// TIA Portal project "INDEXING STATION" (V16)

(* hardware
DEVICE "S7-1200 station_1"  S7-1200 Station
   slot 0: "Rack_0"  S7-1200 Rack  Rack  V1.0
   slot 1: "plc1"  CPU 1214C DC/DC/DC  6ES7 214-1AG40-0XB0  V4.4
DEVICE "ET 200SP station_1"  ET 200SP-Station
   slot 0: "Rack_0"  Rack  6ES5 710-8MAx1
   slot 0: "IO device_1"  IM 155-6 PN/2 HF  6ES7 155-6AU01-0CN0  V4.2
   slot 1: "DI 8x24VDC HF_1"  DI 8x24VDC HF  6ES7 131-6BF00-0CA0  V2.0
      slot 1: "DI 8x24VDC HF_1"  DI 8x24VDC HF
   slot 2: "DI 8x24VDC HF_2"  DI 8x24VDC HF  6ES7 131-6BF00-0CA0  V2.0
      slot 1: "DI 8x24VDC HF_2"  DI 8x24VDC HF
   slot 3: "DI 8x24VDC HF_3"  DI 8x24VDC HF  6ES7 131-6BF00-0CA0  V2.0
      slot 1: "DI 8x24VDC HF_3"  DI 8x24VDC HF
   slot 4: "DQ 8x24VDC/0.5A HF_1"  DQ 8x24VDC/0.5A HF  6ES7 132-6BF00-0CA0  V2.0
      slot 1: "DQ 8x24VDC/0.5A HF_1"  DQ 8x24VDC/0.5A HF
   slot 5: "DQ 8x24VDC/0.5A HF_2"  DQ 8x24VDC/0.5A HF  6ES7 132-6BF00-0CA0  V2.0
      slot 1: "DQ 8x24VDC/0.5A HF_2"  DQ 8x24VDC/0.5A HF
   slot 6: "Server module_1"  Server module  6ES7 193-6PA00-0AA0  V1.1
      slot 1: "Server module_1"  Server module
   slot 127: "BA 2xRJ45"  BA 2xRJ45  6ES7 193-6AR00-0AA0  V0.0
      slot 1: "Port_1"  X1 P1 R  6ES7 193-6AR00-0AA0  V0.0
      slot 2: "Port_2"  X1 P2 R  6ES7 193-6AR00-0AA0  V0.0
*)

// ===== PLC "plc1"  CPU 1214C DC/DC/DC =====

VAR_GLOBAL   // PLC tag table "INPUTS&OUTPUTS_1"
   "S3_START" AT %I0.0 : Bool;
   "S4_STOP" AT %I0.1 : Bool;
   "S5_EMERGENCY_STOP" AT %I0.2 : Bool;
   "S2_OUTPUT_POWER" AT %I0.3 : Bool;
   "S6_RESET" AT %I1.0 : Bool;
   "S_AUTO" AT %I1.1 : Bool;
   "4B1_TRANSFER_CYLINDER_RETRACTED" AT %I1.2 : Bool;
   "4B2_TRANSFER_CYLINDER_EXTENDED" AT %I1.3 : Bool;
   "1B1_LIFT_CYLINDER_RETRACTED" AT %I1.4 : Bool;
   "1B2_LIFT_CYLINDER_EXTENDED" AT %I1.5 : Bool;
   "B3_PART_PRESENT(ORIENTATION_POSITION)" AT %I2.1 : Bool;
   "2B1_ROTATION_CYLINDER_RETRACTED" AT %I2.2 : Bool;
   "2B2_ROTATION_CYLINDER_EXTENDED" AT %I2.3 : Bool;
   "B2_SPOOL_UPPER_PORT" AT %I2.4 : Bool;
   "B4_INDEX_TABLE_HOME" AT %I2.5 : Bool;
   "B5_STEPPER_READY" AT %I2.6 : Bool;
   "B1_PART_PRESENT(INITIAL_POSITION)" AT %I2.7 : Bool;
   "H3_GREEN_ON" AT %Q4.0 : Bool;
   "4M1_EXTEND_TRANSFER" AT %Q4.5 : Bool;
   "1M1_EXTEND_LIFT" AT %Q4.6 : Bool;
   "1M2_RETRACT_LIFT" AT %Q4.7 : Bool;
   "M1_45_STEPPER" AT %Q5.2 : Bool;
   "M1_90_STEPPER" AT %Q5.3 : Bool;
   "3M1_RELEASE_GRIPPER" AT %Q5.4 : Bool;
   "3M2_CLOSE_GRIPPER" AT %Q5.5 : Bool;
   "2M1_EXTEND_ROTATION_CYLINDER" AT %Q5.6 : Bool;
   "2M2_RETRACT_ROTATION_CYLINDER" AT %Q5.7 : Bool;
   "AUTO_MEM" AT %M1.0 : Bool;
   "STOP_MEM" AT %M1.1 : Bool;
   "STEP_2_MEM_ON" AT %M1.2 : Bool;
   "STEP_3&7_MEM_ON" AT %M1.3 : Bool;
   "STEP_4_MEM_ON" AT %M1.4 : Bool;
   "MANUAL_MEM" AT %M1.5 : Bool;
   "STEPPER MEMORY 1" AT %M100.0 : Bool;
   "SM 2" AT %M100.1 : Bool;
   "SM 3" AT %M100.2 : Bool;
   "SM 4" AT %M100.3 : Bool;
   "PART_MEM" AT %M100.4 : Bool;
END_VAR

DATA_BLOCK "STEPS"   // DB1
{ S7_Optimized_Access := 'FALSE' }
VERSION : 0.1
   VAR
      "Current steps" : Int;
   END_VAR
BEGIN
END_DATA_BLOCK

ORGANIZATION_BLOCK "Main"   // OB1, LAD, ProgramCycle
TITLE = "Main Program Sweep (Cycle)"
{ S7_Optimized_Access := 'TRUE' }
VERSION : 0.1
   VAR_INPUT
      Initial_Call : Bool;   // Initial call of this OB
      Remanence : Bool;   // =True, if remanent data are available
   END_VAR
   VAR_TEMP   // added for the SCL form of the ladder/FBD networks
      _w1 : Bool;
   END_VAR
BEGIN

REGION Network 2: START LED ON
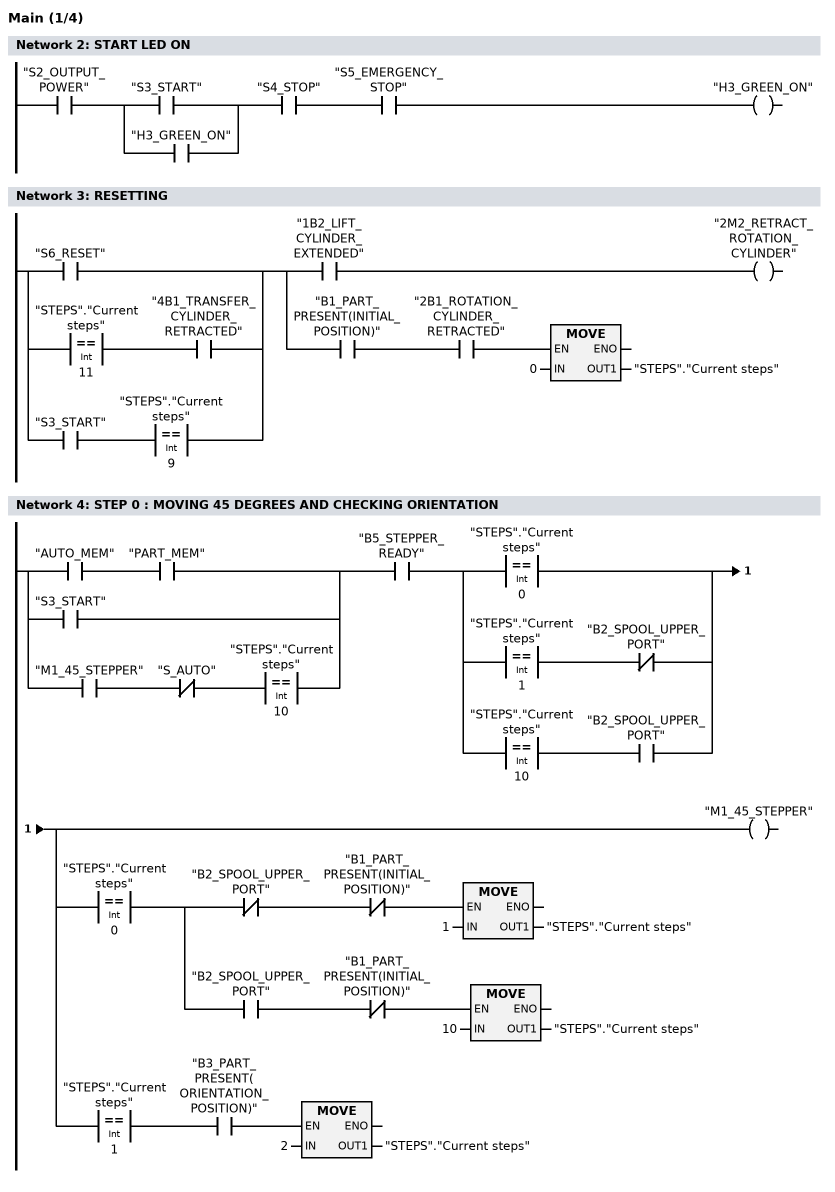
   RUNG wire#powerrail
      Contact( "S2_OUTPUT_POWER" )
      wire#w1
      Contact( "S3_START" )
      wire#w2
      Contact( "S4_STOP" )
      Contact( "S5_EMERGENCY_STOP" )
      Coil( "H3_GREEN_ON" )
   END_RUNG
   RUNG wire#w1
      Contact( "H3_GREEN_ON" )
   END_RUNG wire#w2
   // the same network as SCL:
   "H3_GREEN_ON" := "S2_OUTPUT_POWER" AND ("S3_START" OR "H3_GREEN_ON") AND "S4_STOP" AND "S5_EMERGENCY_STOP";
END_REGION

REGION Network 3: RESETTING
   RUNG wire#powerrail
      Contact( "S6_RESET" )
      wire#w1
      Contact( "1B2_LIFT_CYLINDER_EXTENDED" )
      Coil( "2M2_RETRACT_ROTATION_CYLINDER" )
   END_RUNG
   RUNG wire#powerrail
      { S7_Templates := "SrcType := Int" } EQ_Contact(in1 := "STEPS"."Current steps", in2 := 11)
      Contact( "4B1_TRANSFER_CYLINDER_RETRACTED" )
   END_RUNG wire#w1
   RUNG wire#powerrail
      Contact( "S3_START" )
      { S7_Templates := "SrcType := Int" } EQ_Contact(in1 := "STEPS"."Current steps", in2 := 9)
   END_RUNG wire#w1
   RUNG wire#w1
      Contact( "B1_PART_PRESENT(INITIAL_POSITION)" )
      Contact( "2B1_ROTATION_CYLINDER_RETRACTED" )
      { S7_GenerateENO := "TRUE" } Move(in := 0, out1 => "STEPS"."Current steps")
   END_RUNG
   // the same network as SCL:
   #_w1 := "S6_RESET" OR (("STEPS"."Current steps" = 11) AND "4B1_TRANSFER_CYLINDER_RETRACTED") OR ("S3_START" AND ("STEPS"."Current steps" = 9));
   "2M2_RETRACT_ROTATION_CYLINDER" := #_w1 AND "1B2_LIFT_CYLINDER_EXTENDED";
   IF #_w1 AND "B1_PART_PRESENT(INITIAL_POSITION)" AND "2B1_ROTATION_CYLINDER_RETRACTED" THEN
       "STEPS"."Current steps" := 0;
   END_IF;
END_REGION

REGION Network 4: STEP 0 : MOVING 45 DEGREES AND CHECKING ORIENTATION
   RUNG wire#powerrail
      Contact( "AUTO_MEM" )
      Contact( "PART_MEM" )
      wire#w1
      Contact( "B5_STEPPER_READY" )
      wire#w2
      { S7_Templates := "SrcType := Int" } EQ_Contact(in1 := "STEPS"."Current steps", in2 := 0)
      wire#w3
      Coil( "M1_45_STEPPER" )
   END_RUNG
   RUNG wire#powerrail
      Contact( "S3_START" )
   END_RUNG wire#w1
   RUNG wire#powerrail
      Contact( "M1_45_STEPPER" )
      I_Contact( "S_AUTO" )
      { S7_Templates := "SrcType := Int" } EQ_Contact(in1 := "STEPS"."Current steps", in2 := 10)
   END_RUNG wire#w1
   RUNG wire#w2
      { S7_Templates := "SrcType := Int" } EQ_Contact(in1 := "STEPS"."Current steps", in2 := 1)
      I_Contact( "B2_SPOOL_UPPER_PORT" )
   END_RUNG wire#w3
   RUNG wire#w2
      { S7_Templates := "SrcType := Int" } EQ_Contact(in1 := "STEPS"."Current steps", in2 := 10)
      Contact( "B2_SPOOL_UPPER_PORT" )
   END_RUNG wire#w3
   RUNG wire#w3
      { S7_Templates := "SrcType := Int" } EQ_Contact(in1 := "STEPS"."Current steps", in2 := 0)
      wire#w4
      I_Contact( "B2_SPOOL_UPPER_PORT" )
      I_Contact( "B1_PART_PRESENT(INITIAL_POSITION)" )
      { S7_GenerateENO := "TRUE" } Move(in := 1, out1 => "STEPS"."Current steps")
   END_RUNG
   RUNG wire#w4
      Contact( "B2_SPOOL_UPPER_PORT" )
      I_Contact( "B1_PART_PRESENT(INITIAL_POSITION)" )
      { S7_GenerateENO := "TRUE" } Move(in := 10, out1 => "STEPS"."Current steps")
   END_RUNG
   RUNG wire#w3
      { S7_Templates := "SrcType := Int" } EQ_Contact(in1 := "STEPS"."Current steps", in2 := 1)
      Contact( "B3_PART_PRESENT(ORIENTATION_POSITION)" )
      { S7_GenerateENO := "TRUE" } Move(in := 2, out1 => "STEPS"."Current steps")
   END_RUNG
   // the same network as SCL:
   "M1_45_STEPPER" := (("AUTO_MEM" AND "PART_MEM") OR "S3_START" OR ("M1_45_STEPPER" AND NOT "S_AUTO" AND ("STEPS"."Current steps" = 10))) AND "B5_STEPPER_READY" AND (("STEPS"."Current steps" = 0) OR (("STEPS"."Current steps" = 1) AND NOT "B2_SPOOL_UPPER_PORT") OR (("STEPS"."Current steps" = 10) AND "B2_SPOOL_UPPER_PORT"));
   #_w1 := "M1_45_STEPPER" AND ("STEPS"."Current steps" = 0);
   IF #_w1 AND NOT "B2_SPOOL_UPPER_PORT" AND NOT "B1_PART_PRESENT(INITIAL_POSITION)" THEN
       "STEPS"."Current steps" := 1;
   END_IF;
   IF #_w1 AND "B2_SPOOL_UPPER_PORT" AND NOT "B1_PART_PRESENT(INITIAL_POSITION)" THEN
       "STEPS"."Current steps" := 10;
   END_IF;
   IF "M1_45_STEPPER" AND ("STEPS"."Current steps" = 1) AND "B3_PART_PRESENT(ORIENTATION_POSITION)" THEN
       "STEPS"."Current steps" := 2;
   END_IF;
END_REGION

REGION Network 5: AUTOMATIC_MODE
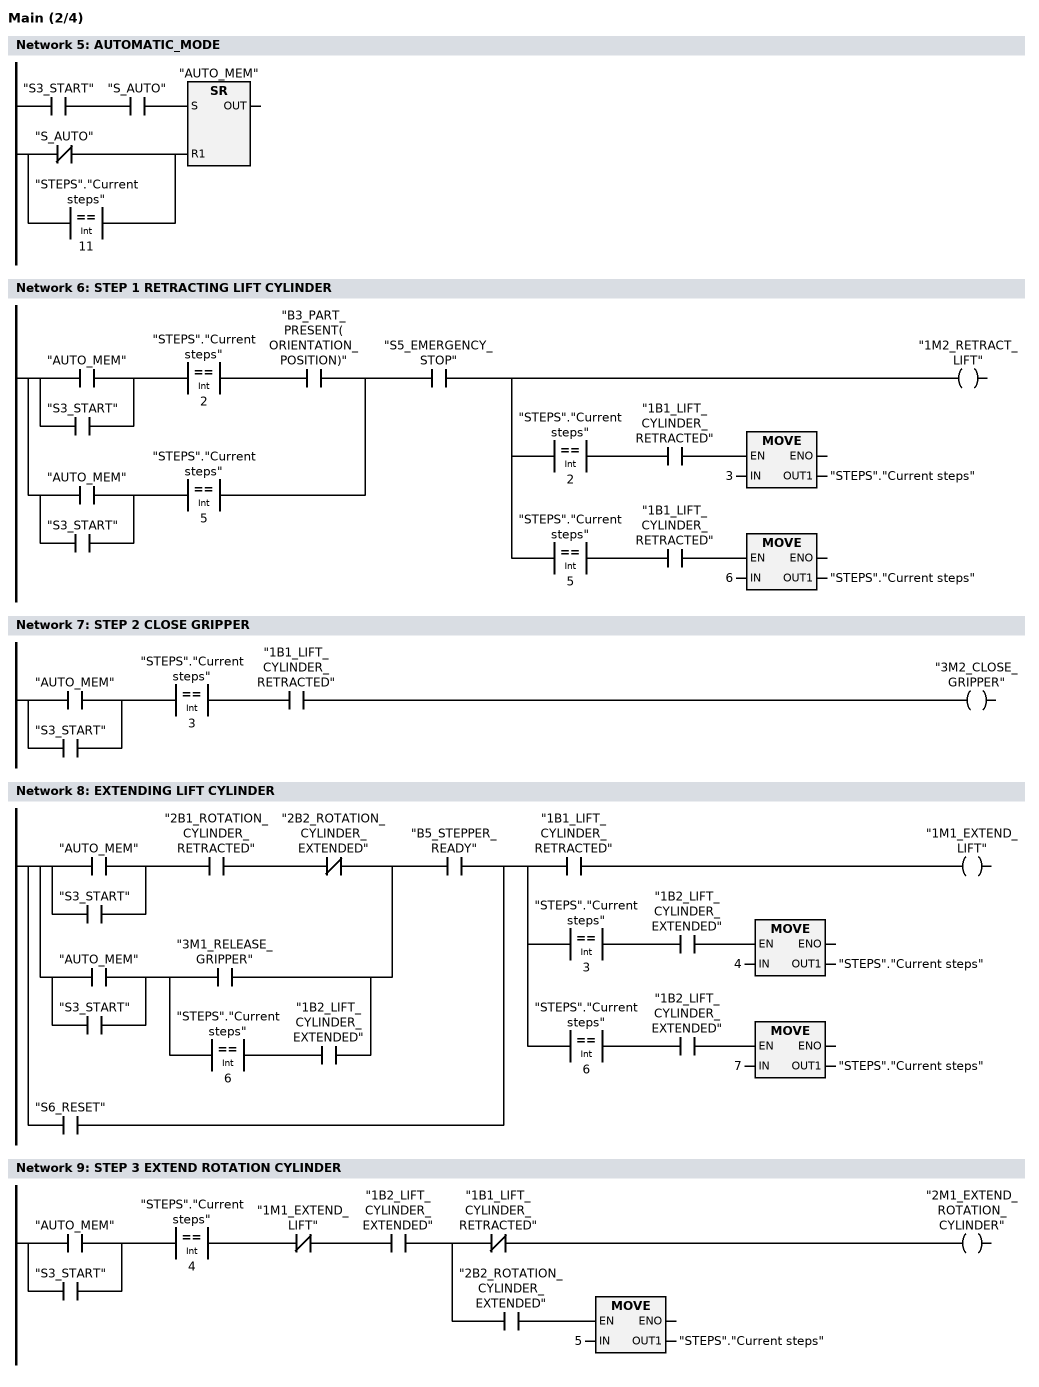
   RUNG wire#powerrail
      Contact( "S3_START" )
      Contact( "S_AUTO" )
      S_SR(operand := "AUTO_MEM", r1 := wire#w1)
   END_RUNG
   RUNG wire#powerrail
      I_Contact( "S_AUTO" )
   END_RUNG wire#w1
   RUNG wire#powerrail
      { S7_Templates := "SrcType := Int" } EQ_Contact(in1 := "STEPS"."Current steps", in2 := 11)
   END_RUNG wire#w1
   // the same network as SCL:
   IF "S3_START" AND "S_AUTO" THEN
       "AUTO_MEM" := TRUE;   // SR flip-flop
   END_IF;
   IF NOT "S_AUTO" OR ("STEPS"."Current steps" = 11) THEN "AUTO_MEM" := FALSE; END_IF;
END_REGION

REGION Network 6: STEP 1 RETRACTING LIFT CYLINDER
   RUNG wire#powerrail
      Contact( "AUTO_MEM" )
      wire#w1
      { S7_Templates := "SrcType := Int" } EQ_Contact(in1 := "STEPS"."Current steps", in2 := 2)
      Contact( "B3_PART_PRESENT(ORIENTATION_POSITION)" )
      wire#w2
      Contact( "S5_EMERGENCY_STOP" )
      wire#w4
      Coil( "1M2_RETRACT_LIFT" )
   END_RUNG
   RUNG wire#powerrail
      Contact( "S3_START" )
   END_RUNG wire#w1
   RUNG wire#powerrail
      Contact( "AUTO_MEM" )
      wire#w3
      { S7_Templates := "SrcType := Int" } EQ_Contact(in1 := "STEPS"."Current steps", in2 := 5)
   END_RUNG wire#w2
   RUNG wire#powerrail
      Contact( "S3_START" )
   END_RUNG wire#w3
   RUNG wire#w4
      { S7_Templates := "SrcType := Int" } EQ_Contact(in1 := "STEPS"."Current steps", in2 := 2)
      Contact( "1B1_LIFT_CYLINDER_RETRACTED" )
      { S7_GenerateENO := "TRUE" } Move(in := 3, out1 => "STEPS"."Current steps")
   END_RUNG
   RUNG wire#w4
      { S7_Templates := "SrcType := Int" } EQ_Contact(in1 := "STEPS"."Current steps", in2 := 5)
      Contact( "1B1_LIFT_CYLINDER_RETRACTED" )
      { S7_GenerateENO := "TRUE" } Move(in := 6, out1 => "STEPS"."Current steps")
   END_RUNG
   // the same network as SCL:
   "1M2_RETRACT_LIFT" := ((("AUTO_MEM" OR "S3_START") AND ("STEPS"."Current steps" = 2) AND "B3_PART_PRESENT(ORIENTATION_POSITION)") OR (("AUTO_MEM" OR "S3_START") AND ("STEPS"."Current steps" = 5))) AND "S5_EMERGENCY_STOP";
   IF "1M2_RETRACT_LIFT" AND ("STEPS"."Current steps" = 2) AND "1B1_LIFT_CYLINDER_RETRACTED" THEN
       "STEPS"."Current steps" := 3;
   END_IF;
   IF "1M2_RETRACT_LIFT" AND ("STEPS"."Current steps" = 5) AND "1B1_LIFT_CYLINDER_RETRACTED" THEN
       "STEPS"."Current steps" := 6;
   END_IF;
END_REGION

REGION Network 7: STEP 2 CLOSE GRIPPER
   RUNG wire#powerrail
      Contact( "AUTO_MEM" )
      wire#w1
      { S7_Templates := "SrcType := Int" } EQ_Contact(in1 := "STEPS"."Current steps", in2 := 3)
      Contact( "1B1_LIFT_CYLINDER_RETRACTED" )
      Coil( "3M2_CLOSE_GRIPPER" )
   END_RUNG
   RUNG wire#powerrail
      Contact( "S3_START" )
   END_RUNG wire#w1
   // the same network as SCL:
   "3M2_CLOSE_GRIPPER" := ("AUTO_MEM" OR "S3_START") AND ("STEPS"."Current steps" = 3) AND "1B1_LIFT_CYLINDER_RETRACTED";
END_REGION

REGION Network 8: EXTENDING LIFT CYLINDER
   RUNG wire#powerrail
      Contact( "AUTO_MEM" )
      wire#w1
      Contact( "2B1_ROTATION_CYLINDER_RETRACTED" )
      I_Contact( "2B2_ROTATION_CYLINDER_EXTENDED" )
      wire#w2
      Contact( "B5_STEPPER_READY" )
      wire#w4
      Contact( "1B1_LIFT_CYLINDER_RETRACTED" )
      Coil( "1M1_EXTEND_LIFT" )
   END_RUNG
   RUNG wire#powerrail
      Contact( "S3_START" )
   END_RUNG wire#w1
   RUNG wire#powerrail
      Contact( "AUTO_MEM" )
      wire#w3
      Contact( "3M1_RELEASE_GRIPPER" )
   END_RUNG wire#w2
   RUNG wire#powerrail
      Contact( "S3_START" )
   END_RUNG wire#w3
   RUNG wire#w3
      { S7_Templates := "SrcType := Int" } EQ_Contact(in1 := "STEPS"."Current steps", in2 := 6)
      Contact( "1B2_LIFT_CYLINDER_EXTENDED" )
   END_RUNG wire#w2
   RUNG wire#powerrail
      Contact( "S6_RESET" )
   END_RUNG wire#w4
   RUNG wire#w4
      { S7_Templates := "SrcType := Int" } EQ_Contact(in1 := "STEPS"."Current steps", in2 := 3)
      Contact( "1B2_LIFT_CYLINDER_EXTENDED" )
      { S7_GenerateENO := "TRUE" } Move(in := 4, out1 => "STEPS"."Current steps")
   END_RUNG
   RUNG wire#w4
      { S7_Templates := "SrcType := Int" } EQ_Contact(in1 := "STEPS"."Current steps", in2 := 6)
      Contact( "1B2_LIFT_CYLINDER_EXTENDED" )
      { S7_GenerateENO := "TRUE" } Move(in := 7, out1 => "STEPS"."Current steps")
   END_RUNG
   // the same network as SCL:
   #_w1 := (((("AUTO_MEM" OR "S3_START") AND "2B1_ROTATION_CYLINDER_RETRACTED" AND NOT "2B2_ROTATION_CYLINDER_EXTENDED") OR (("AUTO_MEM" OR "S3_START") AND ("3M1_RELEASE_GRIPPER" OR (("STEPS"."Current steps" = 6) AND "1B2_LIFT_CYLINDER_EXTENDED")))) AND "B5_STEPPER_READY") OR "S6_RESET";
   "1M1_EXTEND_LIFT" := #_w1 AND "1B1_LIFT_CYLINDER_RETRACTED";
   IF #_w1 AND ("STEPS"."Current steps" = 3) AND "1B2_LIFT_CYLINDER_EXTENDED" THEN
       "STEPS"."Current steps" := 4;
   END_IF;
   IF #_w1 AND ("STEPS"."Current steps" = 6) AND "1B2_LIFT_CYLINDER_EXTENDED" THEN
       "STEPS"."Current steps" := 7;
   END_IF;
END_REGION

REGION Network 9: STEP 3 EXTEND ROTATION CYLINDER
   RUNG wire#powerrail
      Contact( "AUTO_MEM" )
      wire#w1
      { S7_Templates := "SrcType := Int" } EQ_Contact(in1 := "STEPS"."Current steps", in2 := 4)
      I_Contact( "1M1_EXTEND_LIFT" )
      Contact( "1B2_LIFT_CYLINDER_EXTENDED" )
      wire#w2
      I_Contact( "1B1_LIFT_CYLINDER_RETRACTED" )
      Coil( "2M1_EXTEND_ROTATION_CYLINDER" )
   END_RUNG
   RUNG wire#powerrail
      Contact( "S3_START" )
   END_RUNG wire#w1
   RUNG wire#w2
      Contact( "2B2_ROTATION_CYLINDER_EXTENDED" )
      { S7_GenerateENO := "TRUE" } Move(in := 5, out1 => "STEPS"."Current steps")
   END_RUNG
   // the same network as SCL:
   #_w1 := ("AUTO_MEM" OR "S3_START") AND ("STEPS"."Current steps" = 4) AND NOT "1M1_EXTEND_LIFT" AND "1B2_LIFT_CYLINDER_EXTENDED";
   "2M1_EXTEND_ROTATION_CYLINDER" := #_w1 AND NOT "1B1_LIFT_CYLINDER_RETRACTED";
   IF #_w1 AND "2B2_ROTATION_CYLINDER_EXTENDED" THEN "STEPS"."Current steps" := 5; END_IF;
END_REGION

REGION Network 10: STEP 5 RELEASE GRIPPER THEN HEAD TO EXTEND CYLINDER
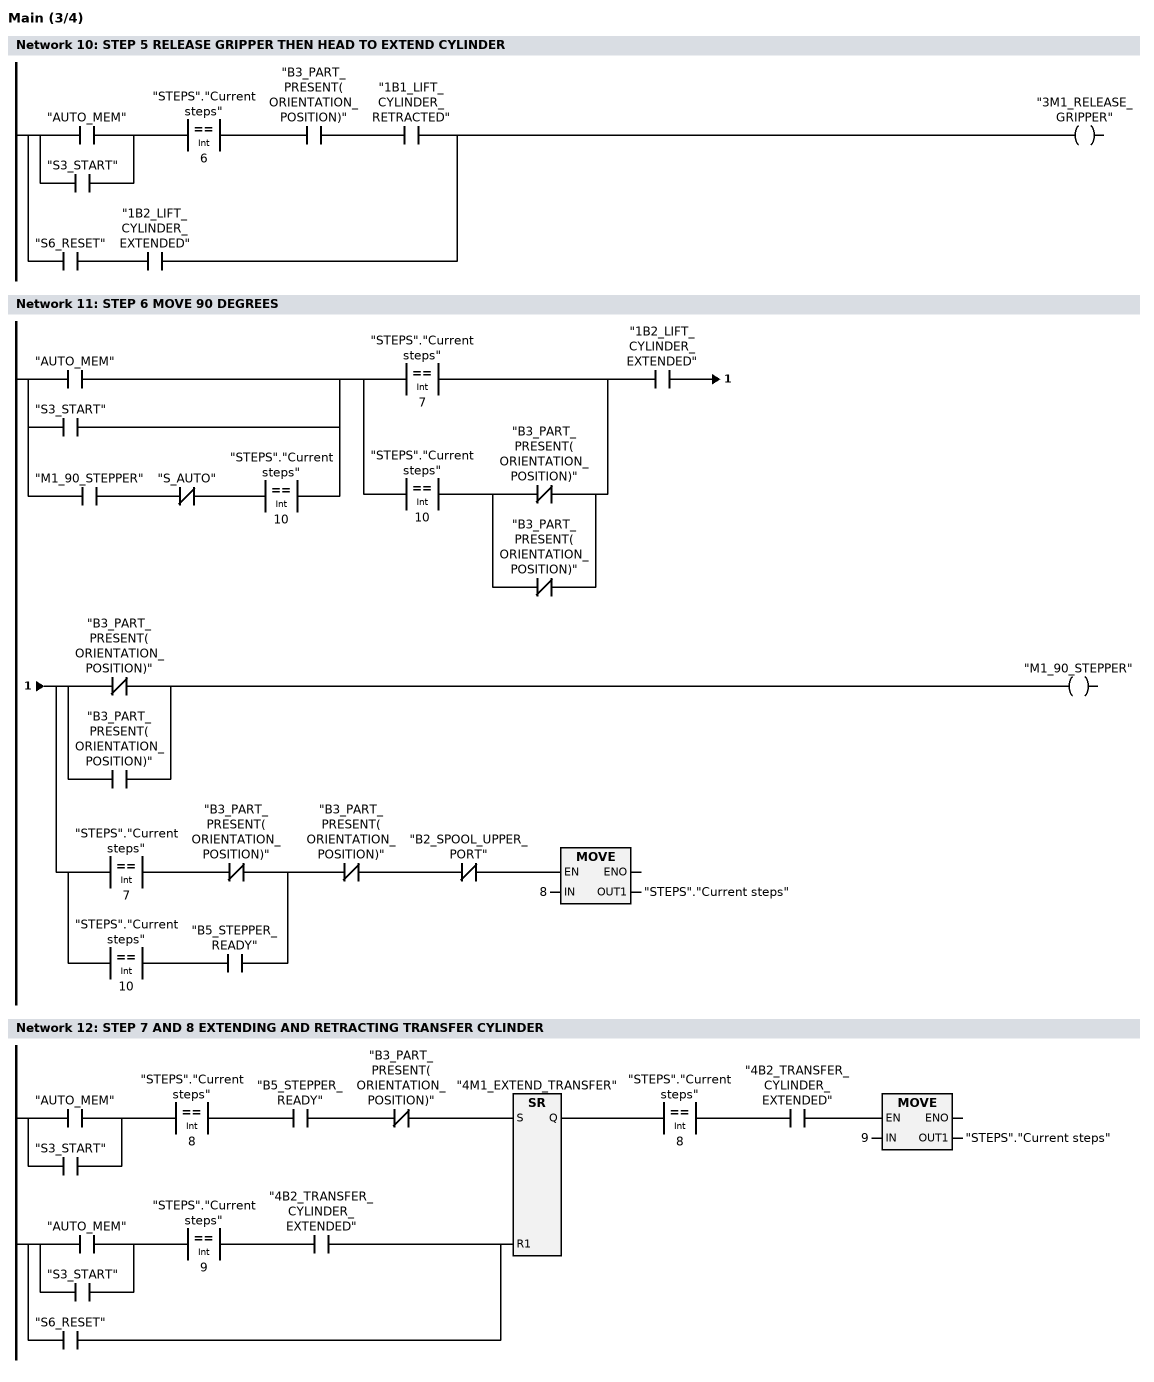
   RUNG wire#powerrail
      Contact( "AUTO_MEM" )
      wire#w1
      { S7_Templates := "SrcType := Int" } EQ_Contact(in1 := "STEPS"."Current steps", in2 := 6)
      Contact( "B3_PART_PRESENT(ORIENTATION_POSITION)" )
      Contact( "1B1_LIFT_CYLINDER_RETRACTED" )
      wire#w2
      Coil( "3M1_RELEASE_GRIPPER" )
   END_RUNG
   RUNG wire#powerrail
      Contact( "S3_START" )
   END_RUNG wire#w1
   RUNG wire#powerrail
      Contact( "S6_RESET" )
      Contact( "1B2_LIFT_CYLINDER_EXTENDED" )
   END_RUNG wire#w2
   // the same network as SCL:
   "3M1_RELEASE_GRIPPER" := (("AUTO_MEM" OR "S3_START") AND ("STEPS"."Current steps" = 6) AND "B3_PART_PRESENT(ORIENTATION_POSITION)" AND "1B1_LIFT_CYLINDER_RETRACTED") OR ("S6_RESET" AND "1B2_LIFT_CYLINDER_EXTENDED");
END_REGION

REGION Network 11: STEP 6 MOVE 90 DEGREES
   RUNG wire#powerrail
      Contact( "AUTO_MEM" )
      wire#w1
      { S7_Templates := "SrcType := Int" } EQ_Contact(in1 := "STEPS"."Current steps", in2 := 7)
      wire#w2
      Contact( "1B2_LIFT_CYLINDER_EXTENDED" )
      wire#w4
      I_Contact( "B3_PART_PRESENT(ORIENTATION_POSITION)" )
      wire#w5
      Coil( "M1_90_STEPPER" )
   END_RUNG
   RUNG wire#powerrail
      Contact( "S3_START" )
   END_RUNG wire#w1
   RUNG wire#powerrail
      Contact( "M1_90_STEPPER" )
      I_Contact( "S_AUTO" )
      { S7_Templates := "SrcType := Int" } EQ_Contact(in1 := "STEPS"."Current steps", in2 := 10)
   END_RUNG wire#w1
   RUNG wire#w1
      { S7_Templates := "SrcType := Int" } EQ_Contact(in1 := "STEPS"."Current steps", in2 := 10)
      wire#w3
      I_Contact( "B3_PART_PRESENT(ORIENTATION_POSITION)" )
   END_RUNG wire#w2
   RUNG wire#w3
      I_Contact( "B3_PART_PRESENT(ORIENTATION_POSITION)" )
   END_RUNG wire#w2
   RUNG wire#w4
      Contact( "B3_PART_PRESENT(ORIENTATION_POSITION)" )
   END_RUNG wire#w5
   RUNG wire#w4
      { S7_Templates := "SrcType := Int" } EQ_Contact(in1 := "STEPS"."Current steps", in2 := 7)
      I_Contact( "B3_PART_PRESENT(ORIENTATION_POSITION)" )
      wire#w6
      I_Contact( "B3_PART_PRESENT(ORIENTATION_POSITION)" )
      I_Contact( "B2_SPOOL_UPPER_PORT" )
      { S7_GenerateENO := "TRUE" } Move(in := 8, out1 => "STEPS"."Current steps")
   END_RUNG
   RUNG wire#w4
      { S7_Templates := "SrcType := Int" } EQ_Contact(in1 := "STEPS"."Current steps", in2 := 10)
      Contact( "B5_STEPPER_READY" )
   END_RUNG wire#w6
   // the same network as SCL:
   #_w1 := ("AUTO_MEM" OR "S3_START" OR ("M1_90_STEPPER" AND NOT "S_AUTO" AND ("STEPS"."Current steps" = 10))) AND (("STEPS"."Current steps" = 7) OR (("STEPS"."Current steps" = 10) AND (NOT "B3_PART_PRESENT(ORIENTATION_POSITION)" OR NOT "B3_PART_PRESENT(ORIENTATION_POSITION)"))) AND "1B2_LIFT_CYLINDER_EXTENDED";
   "M1_90_STEPPER" := #_w1 AND (NOT "B3_PART_PRESENT(ORIENTATION_POSITION)" OR "B3_PART_PRESENT(ORIENTATION_POSITION)");
   IF #_w1 AND ((("STEPS"."Current steps" = 7) AND NOT "B3_PART_PRESENT(ORIENTATION_POSITION)") OR (("STEPS"."Current steps" = 10) AND "B5_STEPPER_READY")) AND NOT "B3_PART_PRESENT(ORIENTATION_POSITION)" AND NOT "B2_SPOOL_UPPER_PORT" THEN
       "STEPS"."Current steps" := 8;
   END_IF;
END_REGION

REGION Network 12: STEP 7 AND 8 EXTENDING AND RETRACTING TRANSFER CYLINDER
   RUNG wire#powerrail
      Contact( "AUTO_MEM" )
      wire#w1
      { S7_Templates := "SrcType := Int" } EQ_Contact(in1 := "STEPS"."Current steps", in2 := 8)
      Contact( "B5_STEPPER_READY" )
      I_Contact( "B3_PART_PRESENT(ORIENTATION_POSITION)" )
      S_SR(operand := "4M1_EXTEND_TRANSFER", r1 := wire#w3)
      { S7_Templates := "SrcType := Int" } EQ_Contact(in1 := "STEPS"."Current steps", in2 := 8)
      Contact( "4B2_TRANSFER_CYLINDER_EXTENDED" )
      { S7_GenerateENO := "TRUE" } Move(in := 9, out1 => "STEPS"."Current steps")
   END_RUNG
   RUNG wire#powerrail
      Contact( "S3_START" )
   END_RUNG wire#w1
   RUNG wire#powerrail
      Contact( "AUTO_MEM" )
      wire#w2
      { S7_Templates := "SrcType := Int" } EQ_Contact(in1 := "STEPS"."Current steps", in2 := 9)
      Contact( "4B2_TRANSFER_CYLINDER_EXTENDED" )
   END_RUNG wire#w3
   RUNG wire#powerrail
      Contact( "S3_START" )
   END_RUNG wire#w2
   RUNG wire#powerrail
      Contact( "S6_RESET" )
   END_RUNG wire#w3
   // the same network as SCL:
   IF ("AUTO_MEM" OR "S3_START") AND ("STEPS"."Current steps" = 8) AND "B5_STEPPER_READY" AND NOT "B3_PART_PRESENT(ORIENTATION_POSITION)" THEN
       "4M1_EXTEND_TRANSFER" := TRUE;   // SR flip-flop
   END_IF;
   IF (("AUTO_MEM" OR "S3_START") AND ("STEPS"."Current steps" = 9) AND "4B2_TRANSFER_CYLINDER_EXTENDED") OR "S6_RESET" THEN
       "4M1_EXTEND_TRANSFER" := FALSE;
   END_IF;
   IF "4M1_EXTEND_TRANSFER" AND ("STEPS"."Current steps" = 8) AND "4B2_TRANSFER_CYLINDER_EXTENDED" THEN
       "STEPS"."Current steps" := 9;
   END_IF;
END_REGION

REGION Network 13: PART MEMORY
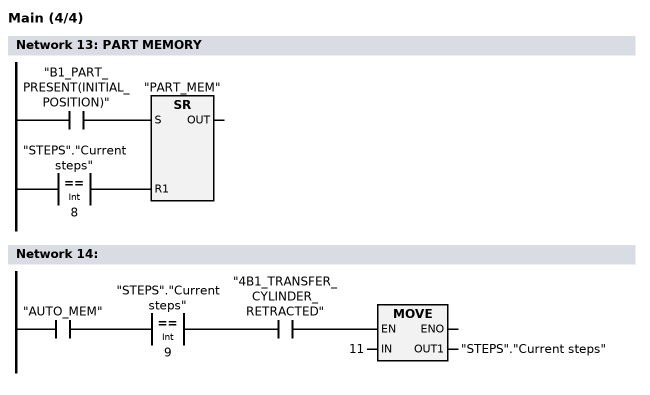
   RUNG wire#powerrail
      Contact( "B1_PART_PRESENT(INITIAL_POSITION)" )
      S_SR(operand := "PART_MEM", r1 := wire#w1)
   END_RUNG
   RUNG wire#powerrail
      { S7_Templates := "SrcType := Int" } EQ_Contact(in1 := "STEPS"."Current steps", in2 := 8)
   END_RUNG wire#w1
   // the same network as SCL:
   IF "B1_PART_PRESENT(INITIAL_POSITION)" THEN
       "PART_MEM" := TRUE;   // SR flip-flop
   END_IF;
   IF "STEPS"."Current steps" = 8 THEN "PART_MEM" := FALSE; END_IF;
END_REGION

REGION Network 14
   RUNG wire#powerrail
      Contact( "AUTO_MEM" )
      { S7_Templates := "SrcType := Int" } EQ_Contact(in1 := "STEPS"."Current steps", in2 := 9)
      Contact( "4B1_TRANSFER_CYLINDER_RETRACTED" )
      { S7_GenerateENO := "TRUE" } Move(in := 11, out1 => "STEPS"."Current steps")
   END_RUNG
   // the same network as SCL:
   IF "AUTO_MEM" AND ("STEPS"."Current steps" = 9) AND "4B1_TRANSFER_CYLINDER_RETRACTED" THEN
       "STEPS"."Current steps" := 11;
   END_IF;
END_REGION
END_ORGANIZATION_BLOCK